FUNCTION_BLOCK FB_DC_MOTOR
VAR_IN_OUT
	Hardware : TYP_DC_MOTOR_HW;
END_VAR
VAR_INPUT
END_VAR
VAR_OUTPUT
	Status : TYP_DC_MOTOR_STATUS;
END_VAR
VAR
	_cmdRun : BOOL;
	_cmdChangeDir : BOOL;
	_cmdNewDir : BOOL;
	PreDelay : TON;
	PostDelay : TON;
END_VAR

IF _cmdRun AND NOT _cmdChangeDir THEN
	IF Hardware.Out.Direction AND Hardware.In.LimitWP THEN
		_cmdRun := FALSE;
	ELSIF NOT Hardware.Out.Direction AND Hardware.In.LimitHP THEN
		_cmdRun := FALSE;
	END_IF;
END_IF;

PreDelay(IN := _cmdChangeDir, PT := T#500MS);
PostDelay(IN := PreDelay.Q, PT := T#500MS);

IF _cmdChangeDir THEN
	THIS^.Hardware.Out.Run := FALSE;
	
	IF PostDelay.Q THEN
		_cmdChangeDir := FALSE;
	ELSIF PreDelay.Q THEN
		THIS^.Hardware.Out.Direction := _cmdNewDir;
	END_IF;
ELSE
	THIS^.Hardware.Out.Run := _cmdRun;
END_IF;

Status.ReachedHP := Hardware.In.LimitHP;
Status.ReachedWP := Hardware.In.LimitWP;

METHOD PUBLIC Run : REFERENCE TO FB_DC_MOTOR
VAR_INPUT
END_VAR
_cmdRun := TRUE;

Run REF= THIS^;
END_METHOD

METHOD PUBLIC SetDirection : REFERENCE TO FB_DC_MOTOR
VAR_INPUT
	Direction : BOOL; // FALSE = forward, TRUE = reverse
END_VAR
VAR
	
END_VAR
_cmdChangeDir := TRUE;
_cmdNewDir := Direction;

SetDirection REF= THIS^;
END_METHOD

METHOD PUBLIC Stop : REFERENCE TO FB_DC_MOTOR
VAR_INPUT
END_VAR
_cmdRun := FALSE;

Stop REF= THIS^;
END_METHOD

END_FUNCTION_BLOCK

(* stored: Version 1.1.0.1, ProductVersion 3.1.4024.12
   POU FB_DC_MOTOR: Id {58c5ca15-8c93-4d48-93fa-508af6307ab4}, SpecialFunc None
   Method Run: Id {075a6a92-2f68-4814-b735-9da70ac4d4f0}
   Method SetDirection: Id {84085ec3-a731-4a3c-a54b-3efb1bd39aa6}
   Method Stop: Id {6074e050-82df-4a55-8220-4f9505d7fb3b} *)
